(*			
	RafalOS
	Rafał Osajda		03.09.2025		TC 4024.66
	Informacja czy w danym elemencie jest jakieś nowe zgłoszenie jeszcze nei wyświetlane i ilosc zgloszen calkowita
*)
TYPE ST_BaseEvents_InformationAboutEventsForHMI :
STRUCT
	bNew				: BOOL;	//nowe
	iQuantity			: INT;	//Ilość
END_STRUCT
END_TYPE

(* stored: Version 1.1.0.1
   DUT ST_BaseEvents_InformationAboutEventsForHMI: Id {cc4a62d2-f4f7-0dcb-3af9-48448cec2c5e} *)
